(* PLC project , CODESYS CODESYS V3.5 SP16 Patch 4 *)
(* stored: creationDateTime 2021-04-28T08:26:31.393707, modificationDateTime 2021-04-27T14:59:42.0020637 *)

FUNCTION_BLOCK ccsSafeCraneNumberSuperv_Test EXTENDS CfUnit.FB_TestSuite
  VAR_INPUT
    in_CraneNoSet1 : WORD;  (* First crane number *)
    in_CraneNoSet2 : WORD;  (* Second crane number *)
  END_VAR
  VAR_OUTPUT
    out_S_CraneNoSupervOk : BOOL;  (* Crane numbers match and are not an empty word *)
    out_S_CraneNo : WORD;  (* A safe crane number. If crane numbers missmatch, this word is set to an empty word *)
  END_VAR
  VAR
    EmptyWord : WORD;
  END_VAR

            FB_Test1();
          

METHOD FB_Test1
  VAR_INPUT
    craneNoSet1 : WORD := 0;  (* First crane number *)
    craneNoSet2 : WORD := 0;  (* Second crane number *)
  END_VAR
  VAR
    Fun : ccsSafeCraneNumberSuperv;
    Result : BOOL;
    ExpectedResult : BOOL := FALSE;
    Condition : BOOL;
  END_VAR
                  TEST('FB_Test1');      																				   (* Naming the test case *)

Fun(in_CraneNoSet1 := craneNoSet1, in_CraneNoSet2 := craneNoSet2, out_S_CraneNoSupervOk => Result);    (* Calling the FB to be tested *)
AssertTrue(Condition := (Result = ExpectedResult),
           Message := 'Result is True');
                                                                                      
TEST_FINISHED();
                
END_METHOD
END_FUNCTION_BLOCK
